FUNCTION_BLOCK F_MUX_4 (* multiplexer *)
  PACKAGE iec61131::selection;
  {SET_ATTRIBUTE(eclipse4diac::core::GenericClassName, 'GEN_F_MUX')}
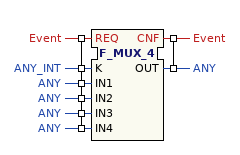
  EVENT_INPUT
    REQ WITH IN1, IN2, IN3, IN4, K; (* Service Request *)
  END_EVENT
  EVENT_OUTPUT
    CNF WITH OUT; (* Confirmation of Requested Service *)
  END_EVENT
  VAR_INPUT
    K : ANY_INT; (* Select one of n inputs *)
    IN1 : ANY; (* Input value 1 *)
    IN2 : ANY; (* Input value 2 *)
    IN3 : ANY; (* Input value 3 *)
    IN4 : ANY; (* Input value 4 *)
  END_VAR
  VAR_OUTPUT
    OUT : ANY; (* IN1 for K = 0, IN2 for K = 1, IN3 for K = 2, IN4 for K = 3 *)
  END_VAR
END_FUNCTION_BLOCK
